// TIA Portal project "CalibrationPanel" (V13)

(* hardware
DEVICE "S7-1200 station_1"  S7-1200 Station
   slot 0: "Rack_0"  Rack  V1.0
   slot 1: "PLC_1"  CPU 1214C DC/DC/DC  6ES7 214-1AG31-0XB0  V3.0
   slot 2: "AI 4x13BIT_1"  6ES7 231-4HD32-0XB0  V2.0
   slot 3: "AQ 2x14BIT_1"  6ES7 232-4HB32-0XB0  V2.0
*)

// ===== PLC "PLC_1"  CPU 1214C DC/DC/DC =====

VAR_GLOBAL   // PLC tag table "plc_tags"
   "System_Byte" AT %MB1 : Byte;
   "FirstScan" AT %M1.0 : Bool;
   "DiagStatusUpdate" AT %M1.1 : Bool;
   "AlwaysTRUE" AT %M1.2 : Bool;
   "AlwaysFALSE" AT %M1.3 : Bool;
   "Clock_Byte" AT %MB0 : Byte;
   "Clock_10Hz" AT %M0.0 : Bool;
   "Clock_5Hz" AT %M0.1 : Bool;
   "Clock_2.5Hz" AT %M0.2 : Bool;
   "Clock_2Hz" AT %M0.3 : Bool;
   "Clock_1.25Hz" AT %M0.4 : Bool;
   "Clock_1Hz" AT %M0.5 : Bool;
   "Clock_0.625Hz" AT %M0.6 : Bool;
   "Clock_0.5Hz" AT %M0.7 : Bool;
END_VAR

VAR_GLOBAL   // PLC tag table "ai_tags"
   "AI_0_IW_Input" AT %IW96 : Int;
   "AI_0_MD_Norm" AT %MD0 : Real;
   "AI_0_MD_Scale" AT %MD4 : Real;
   "AI_1_IW_Input" AT %IW98 : Int;
   "AI_1_MD_Norm" AT %MD20 : Real;
   "AI_1_MD_Scale" AT %MD24 : Real;
   "AI_2_IW_Input" AT %IW100 : Int;
   "AI_2_MD_Norm" AT %MD32 : Real;
   "AI_2_MD_Scale" AT %MD36 : Real;
   "AI_3_IW_Input" AT %IW102 : Int;
   "AI_3_MD_Norm" AT %MD44 : Real;
   "AI_3_MD_Scale" AT %MD48 : Real;
   "AI_4_MD_Norm" AT %MD60 : Real;
   "AI_5_IW_Input" AT %IW66 : Int;
   "AI_4_IW_Input" AT %IW64 : Int;
   "AI_4_MD_Scale" AT %MD64 : Real;
END_VAR

VAR_GLOBAL CONSTANT   // PLC tag table "ai_tags"
   "ZERO_REAL" : Real := 0.00;
   "ZERO_INT" : Int := 0;
   "OUT_RANGE" : Int := 32767;
END_VAR

VAR_GLOBAL   // PLC tag table "ao_tags"
   "AO_0_MD_Norm" AT %MD52 : Real;
   "AO_0_QW_Output" AT %QW112 : Int;
   "AO_1_MD_Norm" AT %MD56 : Real;
   "AO_1_QW_Output" AT %QW114 : Int;
END_VAR

VAR_GLOBAL   // PLC tag table "di_tags"
   "DI_0_I_Input" AT %I0.0 : Bool;
   "DI_1_I_Input" AT %I0.1 : Bool;
   "DI_2_I_Input" AT %I0.2 : Bool;
   "DI_3_I_Input" AT %I0.3 : Bool;
   "DI_4_I_Input" AT %I0.4 : Bool;
END_VAR

VAR_GLOBAL   // PLC tag table "do_tags"
   "DO_0_Q_Output" AT %Q0.0 : Bool;
   "DO_1_Q_Output" AT %Q0.1 : Bool;
   "DO_2_Q_Output" AT %Q0.2 : Bool;
   "DO_3_Q_Output" AT %Q0.3 : Bool;
   "DO_4_Q_Output" AT %Q0.4 : Bool;
   "DO_5_Q_Output" AT %Q0.5 : Bool;
   "DO_6_Q_Output" AT %Q0.6 : Bool;
   "DO_7_Q_Output" AT %Q0.7 : Bool;
END_VAR

DATA_BLOCK "DB_Values"   // DB1
{ S7_Optimized_Access := 'FALSE' }
VERSION : 0.1
   VAR
      AI_0_DB_LRV : Real;
      AI_0_DB_URV : Real;
      AI_0_DB_LPF : Real;
      AI_0_DB_UPF : Real;
      AI_0_DB_Output : Real;
      AI_1_DB_LRV : Real;
      AI_1_DB_URV : Real;
      AI_1_DB_LPF : Real;
      AI_1_DB_UPF : Real;
      AI_1_DB_Output : Real;
      AI_2_DB_Output : Real;
      AI_2_DB_LRV : Real;
      AI_2_DB_URV : Real;
      AI_2_DB_LPF : Real;
      AI_2_DB_UPF : Real;
      AI_3_DB_Output : Real;
      AI_3_DB_LRV : Real;
      AI_3_DB_URV : Real;
      AI_3_DB_LPF : Real;
      AI_3_DB_UPF : Real;
      AO_0_DB_Input : Real;
      AO_1_DB_Input : Real;
      DI_0_DB_Feedback : Bool;
      DI_1_DB_Feedback : Bool;
      DI_2_DB_Feedback : Bool;
      DI_3_DB_Feedback : Bool;
      DI_4_DB_Feedback : Bool;
      DI_5_DB_Feedback : Bool;
      DI_6_DB_Feedback : Bool;
      DI_7_DB_Feedback : Bool;
      DI_8_DB_Feedback : Bool;
      DI_9_DB_Feedback : Bool;
      DI_10_DB_Feedback : Bool;
      DI_11_DB_Feedback : Bool;
      DI_12_DB_Feedback : Bool;
      DI_13_DB_Feedback : Bool;
      DO_0_DB_ActivateOut : Bool;
      DO_1_DB_ActivateOut : Bool;
      DO_2_DB_ActivateOut : Bool;
      DO_3_DB_ActivateOut : Bool;
      DO_4_DB_ActivateOut : Bool;
      DO_5_DB_ActivateOut : Bool;
      DO_6_DB_ActivateOut : Bool;
      DO_7_DB_ActivateOut : Bool;
      DO_8_DB_ActivateOut : Bool;
      DO_9_DB_ActivateOut : Bool;
      AI_2_DB_Output_Feed : Real;
      AI_3_DB_Output_Feed : Real;
      AI_4_DB_LRV : Real;
      AI_4_DB_URV : Real;
      AI_4_DB_LPF : Real;
      AI_4_DB_UPF : Real;
      AI_4_DB_Output : Real;
   END_VAR
BEGIN
END_DATA_BLOCK

ORGANIZATION_BLOCK "Main"   // OB1, LAD, ProgramCycle
TITLE = "Main Program Sweep (Cycle)"
{ S7_Optimized_Access := 'FALSE' }
VERSION : 0.1
BEGIN

REGION Network 1: AI_0
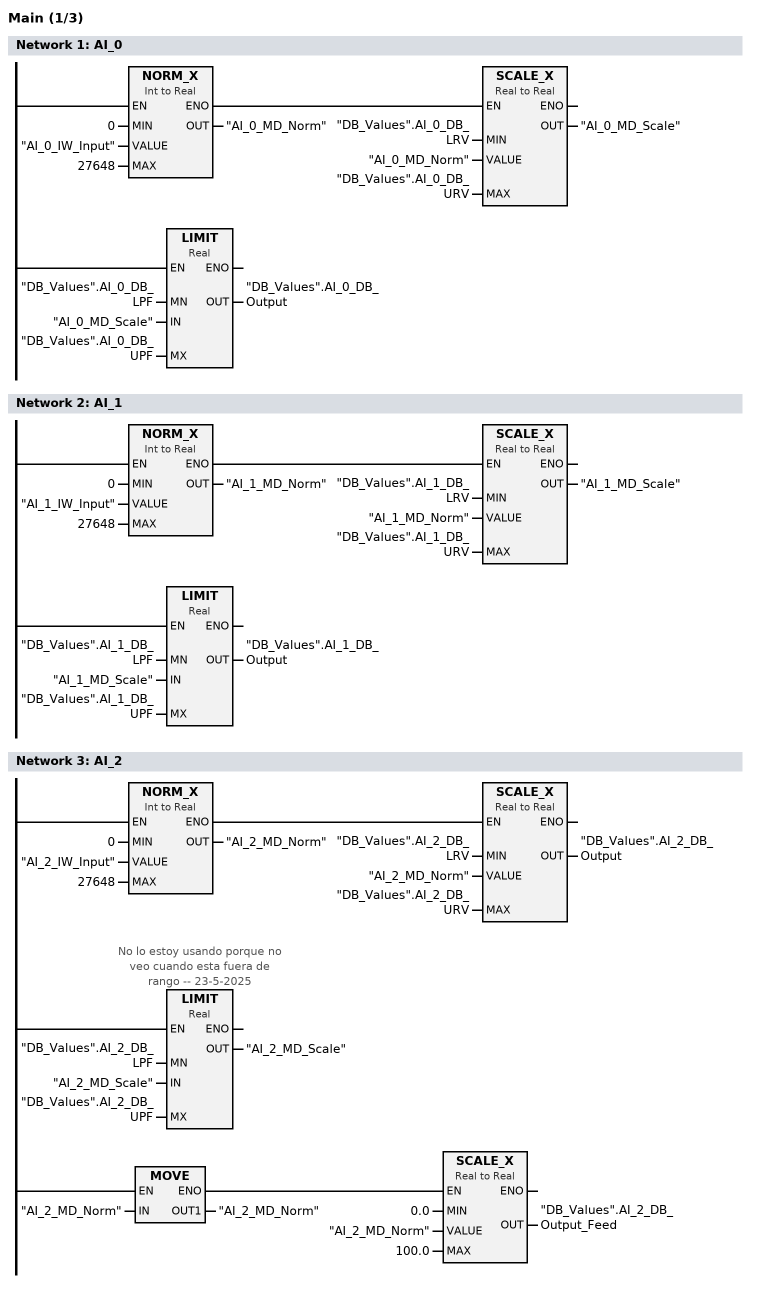
   // ENO of a box is taken as its EN; it also drops when the box reports an error
   "AI_0_MD_Norm" := NORM_X(MIN := 0, VALUE := "AI_0_IW_Input", MAX := 27648);
   "AI_0_MD_Scale" := SCALE_X(MIN := "DB_Values".AI_0_DB_LRV, VALUE := "AI_0_MD_Norm", MAX := "DB_Values".AI_0_DB_URV);
   "DB_Values".AI_0_DB_Output := LIMIT(MN := "DB_Values".AI_0_DB_LPF, IN := "AI_0_MD_Scale", MX := "DB_Values".AI_0_DB_UPF);
END_REGION

REGION Network 2: AI_1
   // ENO of a box is taken as its EN; it also drops when the box reports an error
   "AI_1_MD_Norm" := NORM_X(MIN := 0, VALUE := "AI_1_IW_Input", MAX := 27648);
   "AI_1_MD_Scale" := SCALE_X(MIN := "DB_Values".AI_1_DB_LRV, VALUE := "AI_1_MD_Norm", MAX := "DB_Values".AI_1_DB_URV);
   "DB_Values".AI_1_DB_Output := LIMIT(MN := "DB_Values".AI_1_DB_LPF, IN := "AI_1_MD_Scale", MX := "DB_Values".AI_1_DB_UPF);
END_REGION

REGION Network 3: AI_2
   // ENO of a box is taken as its EN; it also drops when the box reports an error
   "AI_2_MD_Norm" := NORM_X(MIN := 0, VALUE := "AI_2_IW_Input", MAX := 27648);
   "DB_Values".AI_2_DB_Output := SCALE_X(MIN := "DB_Values".AI_2_DB_LRV, VALUE := "AI_2_MD_Norm", MAX := "DB_Values".AI_2_DB_URV);
   "AI_2_MD_Scale" := LIMIT(MN := "DB_Values".AI_2_DB_LPF, IN := "AI_2_MD_Scale", MX := "DB_Values".AI_2_DB_UPF);   // No lo estoy usando porque no veo cuando esta fuera de rango -- 23-5-2025
   "AI_2_MD_Norm" := "AI_2_MD_Norm";
   "DB_Values".AI_2_DB_Output_Feed := SCALE_X(MIN := 0.0, VALUE := "AI_2_MD_Norm", MAX := 100.0);
END_REGION

REGION Network 4: AI_3
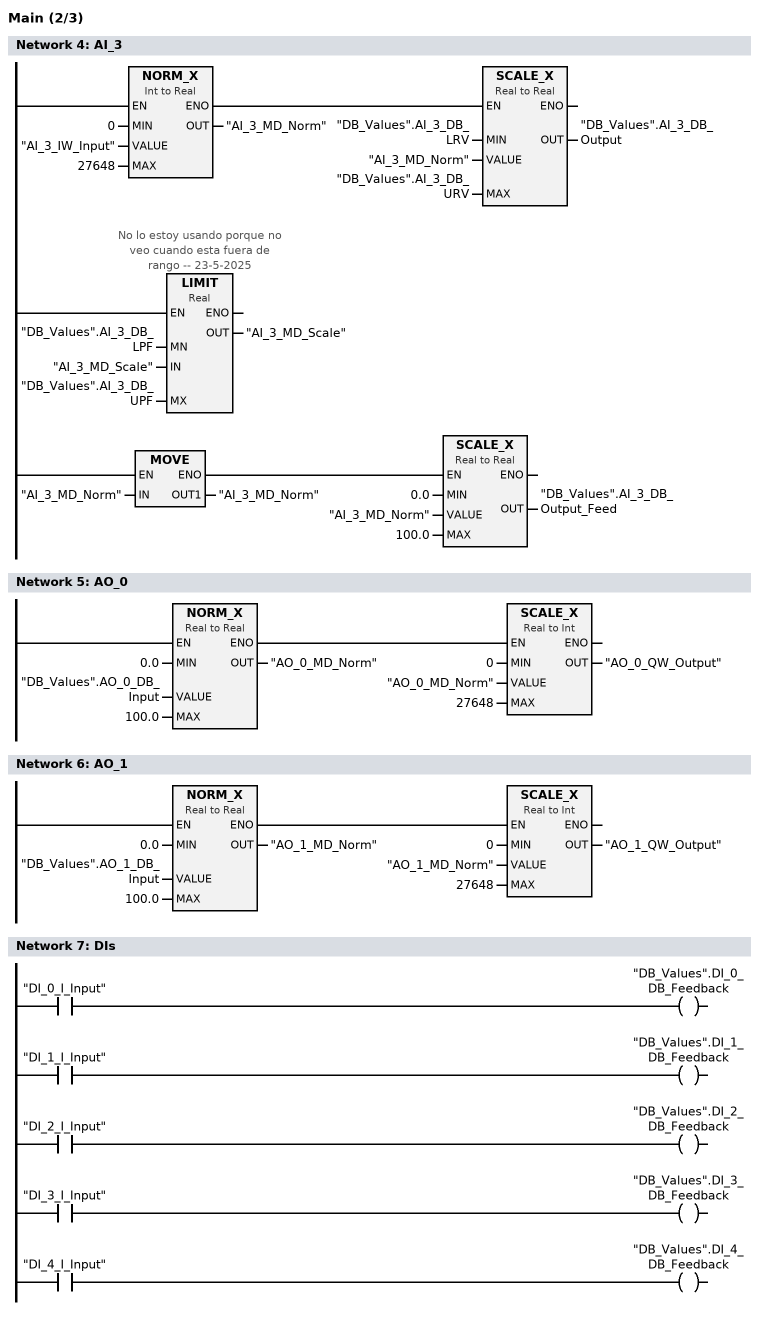
   // ENO of a box is taken as its EN; it also drops when the box reports an error
   "AI_3_MD_Norm" := NORM_X(MIN := 0, VALUE := "AI_3_IW_Input", MAX := 27648);
   "DB_Values".AI_3_DB_Output := SCALE_X(MIN := "DB_Values".AI_3_DB_LRV, VALUE := "AI_3_MD_Norm", MAX := "DB_Values".AI_3_DB_URV);
   "AI_3_MD_Scale" := LIMIT(MN := "DB_Values".AI_3_DB_LPF, IN := "AI_3_MD_Scale", MX := "DB_Values".AI_3_DB_UPF);   // No lo estoy usando porque no veo cuando esta fuera de rango -- 23-5-2025
   "AI_3_MD_Norm" := "AI_3_MD_Norm";
   "DB_Values".AI_3_DB_Output_Feed := SCALE_X(MIN := 0.0, VALUE := "AI_3_MD_Norm", MAX := 100.0);
END_REGION

REGION Network 5: AO_0
   RUNG wire#powerrail
      { S7_Templates := "[SrcType := Real, DestType := Real]"; S7_GenerateENO := "TRUE" } Normalize(min := 0.0, value := "DB_Values".AO_0_DB_Input, max := 100.0, out => "AO_0_MD_Norm")
      { S7_Templates := "[SrcType := Real, DestType := Int]"; S7_GenerateENO := "TRUE" } Scale(min := 0, value := "AO_0_MD_Norm", max := 27648, out => "AO_0_QW_Output")
   END_RUNG
   // the same network as SCL:
   // ENO of a box is taken as its EN; it also drops when the box reports an error
   "AO_0_MD_Norm" := NORM_X(MIN := 0.0, VALUE := "DB_Values".AO_0_DB_Input, MAX := 100.0);
   "AO_0_QW_Output" := SCALE_X(MIN := 0, VALUE := "AO_0_MD_Norm", MAX := 27648);
END_REGION

REGION Network 6: AO_1
   RUNG wire#powerrail
      { S7_Templates := "[SrcType := Real, DestType := Real]"; S7_GenerateENO := "TRUE" } Normalize(min := 0.0, value := "DB_Values".AO_1_DB_Input, max := 100.0, out => "AO_1_MD_Norm")
      { S7_Templates := "[SrcType := Real, DestType := Int]"; S7_GenerateENO := "TRUE" } Scale(min := 0, value := "AO_1_MD_Norm", max := 27648, out => "AO_1_QW_Output")
   END_RUNG
   // the same network as SCL:
   // ENO of a box is taken as its EN; it also drops when the box reports an error
   "AO_1_MD_Norm" := NORM_X(MIN := 0.0, VALUE := "DB_Values".AO_1_DB_Input, MAX := 100.0);
   "AO_1_QW_Output" := SCALE_X(MIN := 0, VALUE := "AO_1_MD_Norm", MAX := 27648);
END_REGION

REGION Network 7: DIs
   RUNG wire#powerrail
      Contact( "DI_0_I_Input" )
      Coil( "DB_Values".DI_0_DB_Feedback )
   END_RUNG
   RUNG wire#powerrail
      Contact( "DI_1_I_Input" )
      Coil( "DB_Values".DI_1_DB_Feedback )
   END_RUNG
   RUNG wire#powerrail
      Contact( "DI_2_I_Input" )
      Coil( "DB_Values".DI_2_DB_Feedback )
   END_RUNG
   RUNG wire#powerrail
      Contact( "DI_3_I_Input" )
      Coil( "DB_Values".DI_3_DB_Feedback )
   END_RUNG
   RUNG wire#powerrail
      Contact( "DI_4_I_Input" )
      Coil( "DB_Values".DI_4_DB_Feedback )
   END_RUNG
   // the same network as SCL:
   "DB_Values".DI_0_DB_Feedback := "DI_0_I_Input";
   "DB_Values".DI_1_DB_Feedback := "DI_1_I_Input";
   "DB_Values".DI_2_DB_Feedback := "DI_2_I_Input";
   "DB_Values".DI_3_DB_Feedback := "DI_3_I_Input";
   "DB_Values".DI_4_DB_Feedback := "DI_4_I_Input";
END_REGION

REGION Network 8: DOs
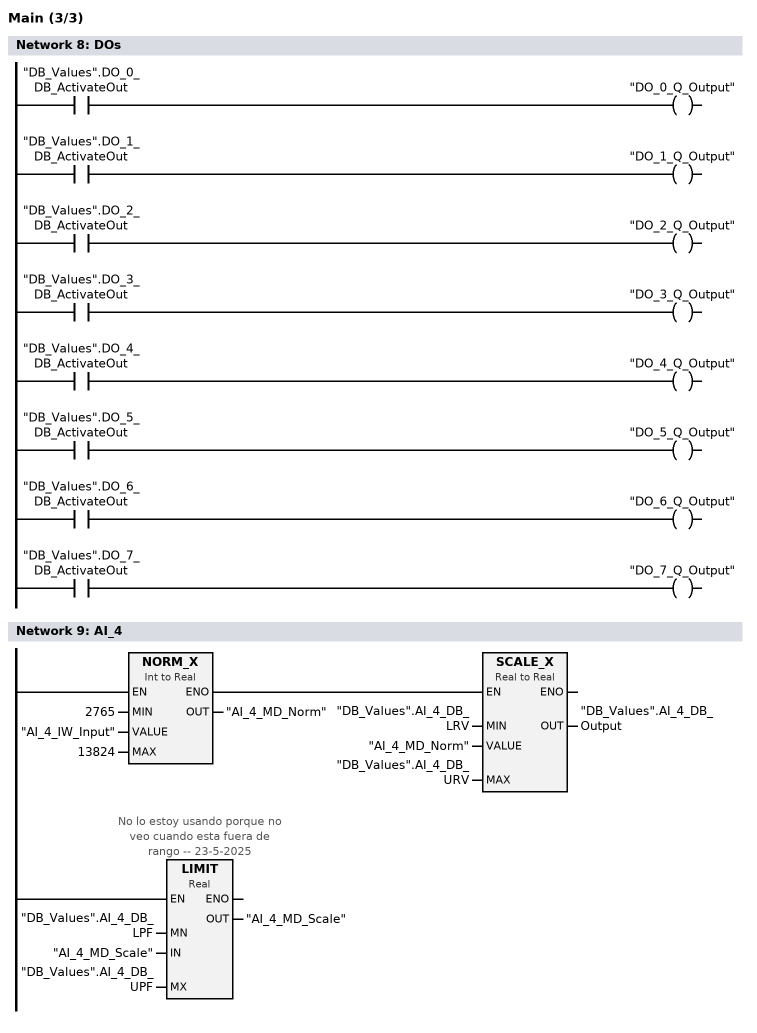
   RUNG wire#powerrail
      Contact( "DB_Values".DO_0_DB_ActivateOut )
      Coil( "DO_0_Q_Output" )
   END_RUNG
   RUNG wire#powerrail
      Contact( "DB_Values".DO_1_DB_ActivateOut )
      Coil( "DO_1_Q_Output" )
   END_RUNG
   RUNG wire#powerrail
      Contact( "DB_Values".DO_2_DB_ActivateOut )
      Coil( "DO_2_Q_Output" )
   END_RUNG
   RUNG wire#powerrail
      Contact( "DB_Values".DO_3_DB_ActivateOut )
      Coil( "DO_3_Q_Output" )
   END_RUNG
   RUNG wire#powerrail
      Contact( "DB_Values".DO_4_DB_ActivateOut )
      Coil( "DO_4_Q_Output" )
   END_RUNG
   RUNG wire#powerrail
      Contact( "DB_Values".DO_5_DB_ActivateOut )
      Coil( "DO_5_Q_Output" )
   END_RUNG
   RUNG wire#powerrail
      Contact( "DB_Values".DO_6_DB_ActivateOut )
      Coil( "DO_6_Q_Output" )
   END_RUNG
   RUNG wire#powerrail
      Contact( "DB_Values".DO_7_DB_ActivateOut )
      Coil( "DO_7_Q_Output" )
   END_RUNG
   // the same network as SCL:
   "DO_0_Q_Output" := "DB_Values".DO_0_DB_ActivateOut;
   "DO_1_Q_Output" := "DB_Values".DO_1_DB_ActivateOut;
   "DO_2_Q_Output" := "DB_Values".DO_2_DB_ActivateOut;
   "DO_3_Q_Output" := "DB_Values".DO_3_DB_ActivateOut;
   "DO_4_Q_Output" := "DB_Values".DO_4_DB_ActivateOut;
   "DO_5_Q_Output" := "DB_Values".DO_5_DB_ActivateOut;
   "DO_6_Q_Output" := "DB_Values".DO_6_DB_ActivateOut;
   "DO_7_Q_Output" := "DB_Values".DO_7_DB_ActivateOut;
END_REGION

REGION Network 9: AI_4
   // ENO of a box is taken as its EN; it also drops when the box reports an error
   "AI_4_MD_Norm" := NORM_X(MIN := 2765, VALUE := "AI_4_IW_Input", MAX := 13824);
   "DB_Values".AI_4_DB_Output := SCALE_X(MIN := "DB_Values".AI_4_DB_LRV, VALUE := "AI_4_MD_Norm", MAX := "DB_Values".AI_4_DB_URV);
   "AI_4_MD_Scale" := LIMIT(MN := "DB_Values".AI_4_DB_LPF, IN := "AI_4_MD_Scale", MX := "DB_Values".AI_4_DB_UPF);   // No lo estoy usando porque no veo cuando esta fuera de rango -- 23-5-2025
END_REGION
END_ORGANIZATION_BLOCK